Staubli VAL3: getValue.pgx

program getValue(string& x_sData (dimensions=1), num& x_nData (dimensions=1), bool& x_bResult (dimensions=1))
  local bool l_bStop
  local string l_sData
  local string l_sString
begin
  do
    l_sString=left(x_sData,1)
    if l_sString!=";" and l_sString!="$"
      l_sData=l_sData+l_sString
    else
      l_bStop=true
    endIf
    x_sData=delete(x_sData,1,0)
    delay(0)
  until l_bStop
  toNum(l_sData,x_nData,x_bResult)
end
